PROGRAM xPlanarRandomSequence
VAR
	Enable			: xPlanarPower;
	Utility			: xPlanarUtility;
	ErrorHandle		: xPlanarErrorHandling;
	MoveSequence	: xPlanarMovements;
	
	Begin			: BOOL;
	
	MainState		: INT;
	Running			: BYTE;
	
	RandomNumGen	: DRAND;
	Seed			: INT := 8729;
	RandomState		: INT;
END_VAR

Enable();
Utility();
ErrorHandle();



Running := Running + 1;

MoveSequence.DefineParameters();

RandomNumGen.Seed := Seed;


CASE MainState OF
		
	0:
		IF Enable.EnableDone THEN
			MainState := 1;
		END_IF	
		
	1:
		MoveSequence.Home(Run := TRUE);
		
		IF MoveSequence.MoveDone THEN
			MainState := 2;
		END_IF
		
	2:
		RandomNumGen();
		RandomState := LREAL_TO_INT(RandomNumGen.Num * 4) + 3;
		MainState := RandomState;
		
	3:
		MoveSequence.SwapPlaces(Run := TRUE);
		
		IF MoveSequence.MoveDone THEN
			MainState := 1;
		END_IF
		
	4:
		MoveSequence.FollowTileEdge(Run := TRUE);
		
		IF MoveSequence.MoveDone THEN
			MainState := 1;
		END_IF	

	5:
		MoveSequence.VaryMoverHeight(Run := TRUE);
		
		IF MoveSequence.MoveDone THEN
			MainState := 1;
		END_IF
		
	6:
		MoveSequence.Tilt(Run := TRUE);
		
		IF MoveSequence.MoveDone THEN
			MainState := 1;
		END_IF
		
	7:
		MoveSequence.Spin(Run := TRUE);
		
		IF MoveSequence.MoveDone THEN
			MainState := 1;
		END_IF
		
END_CASE

END_PROGRAM

(* stored: Version 1.1.0.1, ProductVersion 3.1.4024.12
   POU xPlanarRandomSequence: Id {018c80db-0fff-4570-b60f-32b1bf29accd}, SpecialFunc None *)
